TYPE ref_palletize :
STRUCT
	Pos : ARRAY[1..4] OF ref_xyz ;
	teachingDetail : ref_teachingDetail;
	teachingDetailVels : s_velsXYZ;
END_STRUCT
END_TYPE

(* stored: Version 1.1.0.1, ProductVersion 3.1.4024.11
   DUT ref_palletize: Id {2eed6b72-be6c-4a61-b2b8-89ac0aeab4a5} *)
